FUNCTION_BLOCK FB_Motor
VAR_INPUT
END_VAR
VAR_OUTPUT
END_VAR
VAR
	powerStepper : MC_PowerStepper;
END_VAR

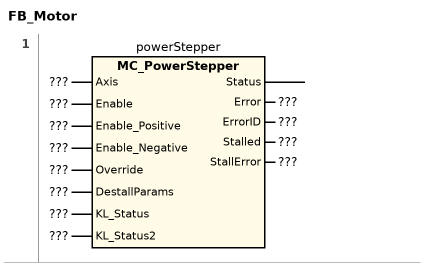
// NETWORK 1
powerStepper(); // MC_PowerStepper

END_FUNCTION_BLOCK

(* stored: Version 1.1.0.1, ProductVersion 3.1.4024.6
   POU FB_Motor: Id {cf0849ea-4cc4-4e7a-a3a4-0cd6c0ed7cdf}, SpecialFunc None *)
